// TwinCAT 3 PLC project ConveyorPLC
// ProgramVersion: 3.1.4026.24
// libraries:
//   Tc2_Standard, * (Beckhoff Automation GmbH)
//   Tc2_System, * (Beckhoff Automation GmbH)
// project tree:
//   GVLs/ GVL.TcGVL, GVL_ModbusIO.TcGVL
//   / PlcTask.TcTTO
//   POUs/ MAIN.TcPOU
// real-time tasks:
//   TASK PlcTask: cycle T#10ms, priority 20, ADS port 350

CONFIGURATION ConveyorPLC
    RESOURCE PLC ON TwinCAT3
        TASK PlcTask(INTERVAL := T#10ms, PRIORITY := 20);
        PROGRAM MAIN WITH PlcTask : MAIN;
    END_RESOURCE
END_CONFIGURATION

// ---- GVLs/GVL.TcGVL
{attribute 'qualified_only'}
VAR_GLOBAL
	mb_Input_Coils      : ARRAY[0..255] OF BOOL; //Modbus coils 32768+
	mb_Output_Coils     : ARRAY[0..255] OF BOOL;
	mb_Input_Registers  : ARRAY[0..255] OF WORD; //Modbus input regs 32768+
	mb_Output_Registers : ARRAY[0..255] OF WORD; //Modbus holding regs 32768+
END_VAR

// ---- GVLs/GVL_ModbusIO.TcGVL
// Modbus I/O boundary - TF6250 maps holding register 32768+n to %MB(2n){attribute 'qualified_only'}
VAR_GLOBAL
	mwSensors   AT %MB0 : WORD; //Webots write: bit0 = entry eye, bit1 = exit eye
	mwActuators AT %MB2 : WORD; //PLC writes:   bit0 = conveyor run
END_VAR

// ---- POUs/MAIN.TcPOU
PROGRAM MAIN
VAR
	nCount : UDINT;
	tBlink :TON;       // timer instance -it has its own memory
	bLight : BOOL;     // the output that will blink
END_VAR

nCount := nCount + 1;

// run the timer; when it expires, toggle the light and restart
tBlink(IN := NOT tBlink.Q, PT := T#500MS);

IF tBlink.Q THEN
	bLight := NOT bLight;
END_IF

GVL_ModbusIO.mwActuators.0 := bLight;
GVL.mb_Output_Registers[0].0 := bLight;

END_PROGRAM
